TYPE TcoUrRoboticsT2OTool :
STRUCT
    {attribute addProperty Name "<#Tool mode#>"}
    ToolMode : USINT;
    {attribute addProperty Name "<#TDI: Tool Digital Inputs#>"}
    TDI_ToolDigitalInputs : USINT;
    {attribute addProperty Name "<#TDO: Tool Digital Outputs#>"}
    TDO_ToolDigitalOutputs : USINT;
    {attribute addProperty Name "<#TAIT: Tool Analog Input Types#>"}
    TAIT_ToolAnalogInputTypes : USINT;
    {attribute addProperty Name "<#Tool analog input [A OR V]#>"}
    ToolAnalogInput : ARRAY[0..1] OF REAL;
    {attribute addProperty Name "<#Tool output voltage [V]#>"}
    ToolOutputVoltage : REAL;
    {attribute addProperty Name "<#Tool current [A]#>"}
    ToolCurrent : REAL;
END_STRUCT
END_TYPE

(* stored: Version 1.1.0.1, ProductVersion 3.1.4024.12
   DUT TcoUrRoboticsT2OTool: Id {ca4244df-d10b-035a-2fe0-4e3e1488d3b9} *)
